VISUALIZATION VISU_AxesExternalSetpointGenerator  // 2x2
END_VISUALIZATION

(* stored: Version 1.1.0.1, ProductVersion 3.1.4018.5
   Visu VISU_AxesExternalSetpointGenerator: Id {f57c73b8-cb13-424b-ba2e-f017f495a089} *)
